// TIA Portal V16 export
// export: Created 2021-09-08T12:46:12.518244Z, ExportSetting WithDefaults, DisplayName Totally Integrated Automation Portal, DisplayVersion V16 Update 3, DisplayName TIA Portal Version Control Interface, DisplayVersion V16 Update 2, DisplayName TIA Portal Openness, DisplayVersion V16 Update 3, DisplayName TIA Portal Teamcenter Gateway, DisplayVersion V16, DisplayName STEP 7 Professional, DisplayVersion V16 Update 3, DisplayName STEP 7 Safety, DisplayVersion V16, DisplayName WinCC Advanced, DisplayVersion V16 Update 3
DATA_BLOCK "AllDigital_DB"   // DB17
VERSION : 0.1
// stored: AutoNumber true, DBAccessibleFromOPCUA true, InstanceOfName AllDigital, InstanceOfType FB
"AllDigital"
   // VAR
   //    FL501 { S7_SetPoint := 'True'} : "DigitalSensorCntrl";
   //    FL901 { S7_SetPoint := 'True'} : "DigitalSensorCntrl";
   //    FL1301 { S7_SetPoint := 'True'} : "DigitalSensorCntrl";
   //    PS901 { S7_SetPoint := 'True'} : "DigitalSensorCntrl";
   //    PS902 { S7_SetPoint := 'True'} : "DigitalSensorCntrl";
   //    PS1301 { S7_SetPoint := 'True'} : "DigitalSensorCntrl";
   //    PS1302 { S7_SetPoint := 'True'} : "DigitalSensorCntrl";
   // END_VAR
BEGIN
END_DATA_BLOCK
